Staubli VAL3: page_Template4.dtx

num nTime = 1
num nKey
num nRefresh
num nView
num nIndex
public string sItems
string sMessage
string sMenu
string sList
string sEvent
bool bButton[8]
bool bLarge
